// TIA Portal V17 export
// export: Created 2025-03-10T12:18:55.0662093Z, ExportSetting WithDefaults, DisplayName Totally Integrated Automation Portal, DisplayVersion V17 Update 8, DisplayName TIA Portal Openness, DisplayVersion V17 Update 8, DisplayName TIA Portal Version Control Interface, DisplayVersion V17, DisplayName SINAMICS Startdrive Advanced, DisplayVersion V17 SP2, DisplayName SINAMICS Startdrive G110M, G120, G120C, G120D, G120P, G115D, DisplayVersion V17 SP2, DisplayName SINAMICS Startdrive G130, G150, S120, S150, SINAMICS MV, S210, DisplayVersion V17 SP2, DisplayName STEP 7 Professional, DisplayVersion V17 Update 8, DisplayName SINUMERIK ONE STEP 7 Toolbox, DisplayVersion V17 Update 12, DisplayName SINUMERIK 840D sl STEP 7 Toolbox, DisplayVersion V17 Update 12, DisplayName STEP 7 Safety, DisplayVersion V17 Update 6, DisplayName WinCC Advanced, DisplayVersion V17 Update 8
FUNCTION_BLOCK "FB22104_TEMPERATURE_SENSOR"   // FB22104, LAD
TITLE = FB22104 TEMPERATURE SENSOR
{ S7_Optimized_Access := 'FALSE' }
VERSION : 0.1
// stored: AutoNumber false, IsIECCheckEnabled false, SetENOAutomatically false, UDAEnableTagReadback false
   VAR_INPUT
      iANALOG_INPUT : Int;
      iCLEAR_LOG : Bool;
   END_VAR
   VAR_OUTPUT
      oERROR_LIMIT : Bool;
      oWARNING_LIMIT : Bool;
   END_VAR
   VAR DB_SPECIFIC
      OUTPUT : Struct
         VALUE : Real;
      END_STRUCT;
      INPUT_SETTINGS : Struct
         MAX_INPUT_VALUE : Real;
         IS_ANALOG_VALUE : Bool;
         UNIT_NUMBER : Int;
         HOPPER_NUMBER : Int;
      END_STRUCT;
      ALARMS_SETTINGS : Struct
         WARN_LIM_HIGH : Real;
         ERROR_LIM_HIGH : Real;
         WARN_LIM_LOW : Real;
         ERROR_LIM_LOW : Real;
         ERROR_CONFIGURATION : Bool;
      END_STRUCT;
      LOG : Struct
         MAX_TEMP_DATE : Date_And_Time;
         MAX_TEMP : Real;
      END_STRUCT;
      INTERNAL : Struct
         ERROR_CODE_T : Int;
         AUX : Bool;
      END_STRUCT;
   END_VAR
   VAR_TEMP
      DB_NUMBER : DInt;
      RET_VAL : Int;
      ZERO : Int;
      CONV_VALUE : DInt;
      NORM_VALUE : Real;
   END_VAR
   VAR_TEMP   // added for the SCL form of the ladder/FBD networks
      _w1 : Bool;
      _w2 : Bool;
   END_VAR
BEGIN

NETWORK
TITLE = READ INSTANCE DB NUMBER
      L     DINO;
      +     10#800000;
      T     #DB_NUMBER;

REGION Network 2: CONVERT, NORM AND SCALE ANALOG INPUT / Scaling temperature value from the sensor
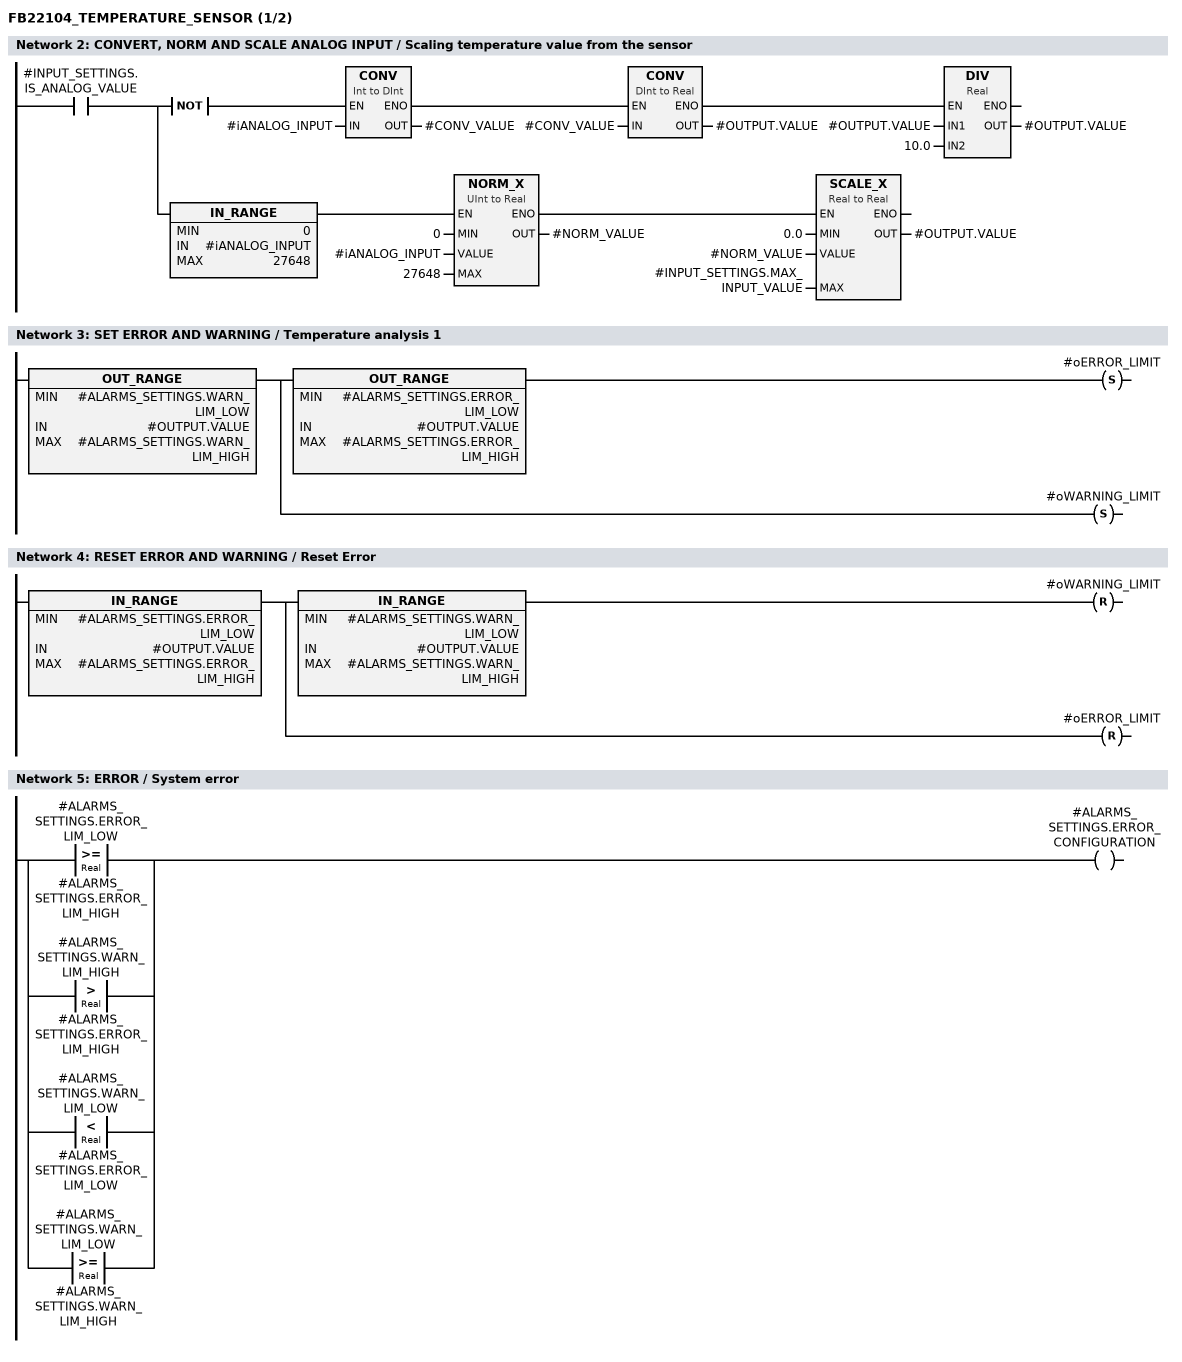
   RUNG wire#powerrail
      Contact( #INPUT_SETTINGS.IS_ANALOG_VALUE )
      wire#w1
      Not()
      { S7_Templates := "[SrcType := Int, DestType := DInt]"; S7_GenerateENO := "TRUE" } Convert(in := #iANALOG_INPUT, out => #CONV_VALUE)
      { S7_Templates := "[SrcType := DInt, DestType := Real]"; S7_GenerateENO := "TRUE" } Convert(in := #CONV_VALUE, out => #OUTPUT.VALUE)
      { S7_Templates := "SrcType := Real"; S7_GenerateENO := "TRUE" } Div(in1 := #OUTPUT.VALUE, in2 := 10.0, out => #OUTPUT.VALUE)
   END_RUNG
   RUNG wire#w1
      { S7_Templates := "SrcType := Int" } InRange(min := 0, in := #iANALOG_INPUT, max := 27648)
      { S7_Templates := "[SrcType := UInt, DestType := Real]" } Normalize(min := 0, value := #iANALOG_INPUT, max := 27648, out => #NORM_VALUE)
      { S7_Templates := "[SrcType := Real, DestType := Real]" } Scale(min := 0.0, value := #NORM_VALUE, max := #INPUT_SETTINGS.MAX_INPUT_VALUE, out => #OUTPUT.VALUE)
   END_RUNG
   // the same network as SCL:
   // ENO of a box is taken as its EN; it also drops when the box reports an error
   IF NOT #INPUT_SETTINGS.IS_ANALOG_VALUE THEN
       #CONV_VALUE := INT_TO_DINT(#iANALOG_INPUT);
       #OUTPUT.VALUE := DINT_TO_REAL(#CONV_VALUE);
       #OUTPUT.VALUE := #OUTPUT.VALUE / 10.0;
   END_IF;
   IF #INPUT_SETTINGS.IS_ANALOG_VALUE AND (0 <= #iANALOG_INPUT) AND (#iANALOG_INPUT <= 27648) THEN
       #NORM_VALUE := NORM_X(MIN := 0, VALUE := #iANALOG_INPUT, MAX := 27648);
       #OUTPUT.VALUE := SCALE_X(MIN := 0.0, VALUE := #NORM_VALUE, MAX := #INPUT_SETTINGS.MAX_INPUT_VALUE);
   END_IF;
END_REGION

REGION Network 3: SET ERROR AND WARNING / Temperature analysis 1
   #_w1 := (#OUTPUT.VALUE < #ALARMS_SETTINGS.WARN_LIM_LOW) OR (#OUTPUT.VALUE > #ALARMS_SETTINGS.WARN_LIM_HIGH);
   IF #_w1 AND ((#OUTPUT.VALUE < #ALARMS_SETTINGS.ERROR_LIM_LOW) OR (#OUTPUT.VALUE > #ALARMS_SETTINGS.ERROR_LIM_HIGH)) THEN
       #oERROR_LIMIT := TRUE;
   END_IF;
   IF #_w1 THEN #oWARNING_LIMIT := TRUE; END_IF;
END_REGION

REGION Network 4: RESET ERROR AND WARNING / Reset Error
   RUNG wire#powerrail
      { S7_Templates := "SrcType := Real" } InRange(min := #ALARMS_SETTINGS.ERROR_LIM_LOW, in := #OUTPUT.VALUE, max := #ALARMS_SETTINGS.ERROR_LIM_HIGH)
      wire#w1
      { S7_Templates := "SrcType := Real" } InRange(min := #ALARMS_SETTINGS.WARN_LIM_LOW, in := #OUTPUT.VALUE, max := #ALARMS_SETTINGS.WARN_LIM_HIGH)
      R_Coil( #oWARNING_LIMIT )
   END_RUNG
   RUNG wire#w1
      R_Coil( #oERROR_LIMIT )
   END_RUNG
   // the same network as SCL:
   #_w1 := (#ALARMS_SETTINGS.ERROR_LIM_LOW <= #OUTPUT.VALUE) AND (#OUTPUT.VALUE <= #ALARMS_SETTINGS.ERROR_LIM_HIGH);
   IF #_w1 AND (#ALARMS_SETTINGS.WARN_LIM_LOW <= #OUTPUT.VALUE) AND (#OUTPUT.VALUE <= #ALARMS_SETTINGS.WARN_LIM_HIGH) THEN
       #oWARNING_LIMIT := FALSE;
   END_IF;
   IF #_w1 THEN #oERROR_LIMIT := FALSE; END_IF;
END_REGION

REGION Network 5: ERROR / System error
   RUNG wire#powerrail
      { S7_Templates := "SrcType := Real" } GE_Contact(in1 := #ALARMS_SETTINGS.ERROR_LIM_LOW, in2 := #ALARMS_SETTINGS.ERROR_LIM_HIGH)
      wire#w1
      Coil( #ALARMS_SETTINGS.ERROR_CONFIGURATION )
   END_RUNG
   RUNG wire#powerrail
      { S7_Templates := "SrcType := Real" } GT_Contact(in1 := #ALARMS_SETTINGS.WARN_LIM_HIGH, in2 := #ALARMS_SETTINGS.ERROR_LIM_HIGH)
   END_RUNG wire#w1
   RUNG wire#powerrail
      { S7_Templates := "SrcType := Real" } LT_Contact(in1 := #ALARMS_SETTINGS.WARN_LIM_LOW, in2 := #ALARMS_SETTINGS.ERROR_LIM_LOW)
   END_RUNG wire#w1
   RUNG wire#powerrail
      { S7_Templates := "SrcType := Real" } GE_Contact(in1 := #ALARMS_SETTINGS.WARN_LIM_LOW, in2 := #ALARMS_SETTINGS.WARN_LIM_HIGH)
   END_RUNG wire#w1
   // the same network as SCL:
   #ALARMS_SETTINGS.ERROR_CONFIGURATION := (#ALARMS_SETTINGS.ERROR_LIM_LOW >= #ALARMS_SETTINGS.ERROR_LIM_HIGH) OR (#ALARMS_SETTINGS.WARN_LIM_HIGH > #ALARMS_SETTINGS.ERROR_LIM_HIGH) OR (#ALARMS_SETTINGS.WARN_LIM_LOW < #ALARMS_SETTINGS.ERROR_LIM_LOW) OR (#ALARMS_SETTINGS.WARN_LIM_LOW >= #ALARMS_SETTINGS.WARN_LIM_HIGH);
END_REGION

REGION Network 6: SAVE MAX VALUES TO LOG / Maximum temperature value
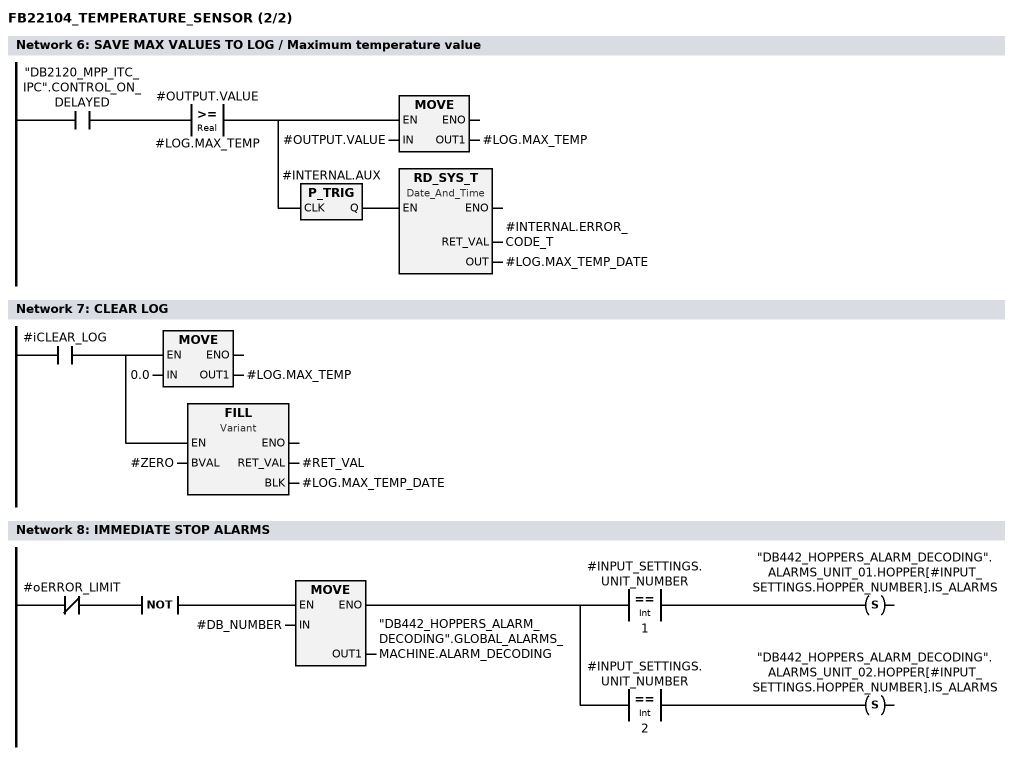
   RUNG wire#powerrail
      Contact( "DB2120_MPP_ITC_IPC".CONTROL_ON_DELAYED )
      { S7_Templates := "SrcType := Real" } GE_Contact(in1 := #OUTPUT.VALUE, in2 := #LOG.MAX_TEMP)
      wire#w1
      { S7_GenerateENO := "TRUE" } Move(in := #OUTPUT.VALUE, out1 => #LOG.MAX_TEMP)
   END_RUNG
   RUNG wire#w1
      P_Trig( #INTERNAL.AUX )
      { S7_Templates := "date_type := Date_And_Time" } RD_SYS_T(RET_VAL => #INTERNAL.ERROR_CODE_T, OUT => #LOG.MAX_TEMP_DATE)
   END_RUNG
   // the same network as SCL:
   #_w1 := "DB2120_MPP_ITC_IPC".CONTROL_ON_DELAYED AND (#OUTPUT.VALUE >= #LOG.MAX_TEMP);
   IF #_w1 THEN #LOG.MAX_TEMP := #OUTPUT.VALUE; END_IF;
   #_w2 := #_w1 AND NOT #INTERNAL.AUX;   // rising edge
   #INTERNAL.AUX := #_w1;
   IF #_w2 THEN #INTERNAL.ERROR_CODE_T := RD_SYS_T(OUT => #LOG.MAX_TEMP_DATE); END_IF;
END_REGION

REGION Network 7: CLEAR LOG
   RUNG wire#powerrail
      Contact( #iCLEAR_LOG )
      wire#w1
      { S7_GenerateENO := "TRUE" } Move(in := 0.0, out1 => #LOG.MAX_TEMP)
   END_RUNG
   RUNG wire#w1
      { S7_Templates := "ptr_type := Variant" } FILL(BVAL := #ZERO, RET_VAL => #RET_VAL, BLK => #LOG.MAX_TEMP_DATE)
   END_RUNG
   // the same network as SCL:
   IF #iCLEAR_LOG THEN
       #LOG.MAX_TEMP := 0.0;
       #RET_VAL := FILL(BVAL := #ZERO, BLK => #LOG.MAX_TEMP_DATE);
   END_IF;
END_REGION

REGION Network 8: IMMEDIATE STOP ALARMS
   RUNG wire#powerrail
      I_Contact( #oERROR_LIMIT )
      Not()
      { S7_GenerateENO := "TRUE" } Move(in := #DB_NUMBER, out1 => "DB442_HOPPERS_ALARM_DECODING".GLOBAL_ALARMS_MACHINE.ALARM_DECODING)
      wire#w1
      { S7_Templates := "SrcType := Int" } EQ_Contact(in1 := #INPUT_SETTINGS.UNIT_NUMBER, in2 := 1)
      S_Coil( "DB442_HOPPERS_ALARM_DECODING".ALARMS_UNIT_01.HOPPER[#INPUT_SETTINGS.HOPPER_NUMBER].IS_ALARMS )
   END_RUNG
   RUNG wire#w1
      { S7_Templates := "SrcType := Int" } EQ_Contact(in1 := #INPUT_SETTINGS.UNIT_NUMBER, in2 := 2)
      S_Coil( "DB442_HOPPERS_ALARM_DECODING".ALARMS_UNIT_02.HOPPER[#INPUT_SETTINGS.HOPPER_NUMBER].IS_ALARMS )
   END_RUNG
   // the same network as SCL:
   // ENO of a box is taken as its EN; it also drops when the box reports an error
   IF NOT (NOT #oERROR_LIMIT) THEN
       "DB442_HOPPERS_ALARM_DECODING".GLOBAL_ALARMS_MACHINE.ALARM_DECODING := #DB_NUMBER;
   END_IF;
   IF NOT (NOT #oERROR_LIMIT) AND (#INPUT_SETTINGS.UNIT_NUMBER = 1) THEN
       "DB442_HOPPERS_ALARM_DECODING".ALARMS_UNIT_01.HOPPER[#INPUT_SETTINGS.HOPPER_NUMBER].IS_ALARMS := TRUE;
   END_IF;
   IF NOT (NOT #oERROR_LIMIT) AND (#INPUT_SETTINGS.UNIT_NUMBER = 2) THEN
       "DB442_HOPPERS_ALARM_DECODING".ALARMS_UNIT_02.HOPPER[#INPUT_SETTINGS.HOPPER_NUMBER].IS_ALARMS := TRUE;
   END_IF;
END_REGION
END_FUNCTION_BLOCK
